RoboDK station: AE1222-2021-GROUP-E09H-RobotMotionPlan.rdk

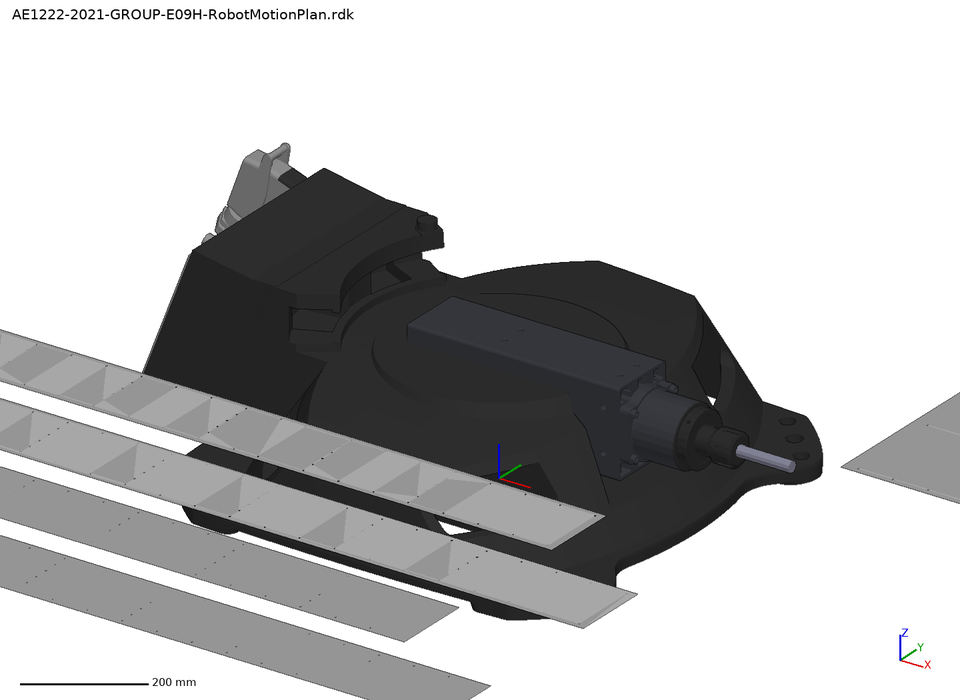
[picture v0: the station drawn from its stored meshes, robots at their saved joint values, targets as dots, program paths as lines]
Station Final (saved by RoboDK 5.2.3). Poses are relative to the parent item; angles as X-Y-Z fixed-axis rotations.
  - frame KUKA KR 210 R2700 extra Base at (0, 0, 0) mm
    - robot KUKA KR 210 R2700 extra: 6 axes, payload 210 kg, reach 2696 mm, repeatability 0.06 mm, weight 1068 kg
        joint limits [-185, -140, -120, -350, -125, -350] to [185, -5, 155, 350, 125, 350]; home [0, -90, 90, 0, 0, 0]; saved at [81.28, -116.082, 145.473, 263.789, 78.817, -240.018]
      - tool Spindle, TCP at (557.2, 0, 176) mm, rotated rx 0 ry 90 rz 0 deg, size 692.9 x 170 x 256 mm
  - Python program Plan, spread panels (listed below)
  - object Panel_Root_Bottom at (1000, 901.6, 500) mm, rotated rx 180 ry 0 rz 0 deg, size 1500 x 400 x 0.8 mm, geometry from Panel_Root_Bottom.stl
  - object Panel_Root_Top at (1000, 1400, 500) mm, rotated rx 180 ry 0 rz 0 deg, size 1500 x 400 x 0.8 mm, geometry from Panel_Root_Top.stl
  - object Panel_Tip - Bottom at (1000, 0, 500) mm, rotated rx 180 ry 0 rz -180 deg, size 1500 x 400 x 0.8 mm, geometry from Panel_Tip - Bottom.stl
  - object Panel_Tip - Top at (1000, -500, 500) mm, rotated rx 180 ry 0 rz -180 deg, size 1500 x 400 x 0.8 mm, geometry from Panel_Tip - Top.stl
  - object Side_Panel_Root_Long at (-500, -1600, 500) mm, rotated rx 0 ry -90 rz -90 deg, size 0.8 x 1500 x 148.4 mm, geometry from Side_Panel_Root_Long.stl
  - object Side_Panel_Root_Short at (-500, -1400, 500) mm, rotated rx 0 ry -90 rz -90 deg, size 0.8 x 1300 x 148.4 mm, geometry from Side_Panel_Root_Short.stl
  - object Side_Panel_Tip_Long at (-500, -1200, 500) mm, rotated rx 0 ry 90 rz 90 deg, size 0.8 x 1500 x 148.4 mm, geometry from Side_Panel_Tip_Long.stl
  - object Side_Panel_Tip_Short at (-500, -1000, 500) mm, rotated rx 0 ry 90 rz 90 deg, size 0.8 x 1300 x 148.4 mm, geometry from Side_Panel_Tip_Short.stl

--- Python program Plan, spread panels ---
from robolink import *
from robodk import *
import time




data = open('AE1222-2021-GROUP-E09H-CoordinateFile-PanelRootBottom.txt')






# read table and get rid of fat
x = 1000
y = 1000
z = 500


table = []
test = []

for line in data:
    row = line.split('\t')
    for i in range(7):
        del row[-1]
    res = [float(i) for i in row]
    res[0] += x
    res[1] += y
    res[2] += z
    table.append(res)
print(table)




RDK = Robolink()


RDK.Render(False)


list_items = RDK.ItemList()
for item in list_items:
    if item.Name().startswith('Auto'):
        item.Delete()


robot = RDK.ItemUserPick('Select a robot', ITEM_TYPE_ROBOT)
robot.setSpeed(500)

RDK.Render(True)


if not robot.Valid():
    quit()


reference = robot.Parent()


robot.setPoseFrame(reference)


pose_ref = robot.Pose()
print(Pose_2_TxyzRxyz(pose_ref))

pose_i = pose_ref
pose_i.setPos(table[0])
robot.MoveJ(pose_i)

for i in range(len(table)-1):

    pose_i = pose_ref
    pose_i.setPos(table[i+1])


    robot.MoveL(pose_i)


data = open('AE1222-2021-GROUP-E09H-CoordinateFile-PanelRootTop.txt')






# read table and get rid of fat
x = 1000
y = 500
z = 500


table = []
test = []

for line in data:
    row = line.split('\t')
    for i in range(7):
        del row[-1]
    res = [float(i) for i in row]
    res[0] += x
    res[1] += y
    res[2] += z
    table.append(res)
print(table)




RDK = Robolink()


RDK.Render(False)


list_items = RDK.ItemList()
for item in list_items:
    if item.Name().startswith('Auto'):
        item.Delete()


robot = RDK.ItemUserPick('Select a robot', ITEM_TYPE_ROBOT)


RDK.Render(True)


if not robot.Valid():
    quit()


reference = robot.Parent()


robot.setPoseFrame(reference)


pose_ref = robot.Pose()
print(Pose_2_TxyzRxyz(pose_ref))





for i in range(len(table)):

    pose_i = pose_ref
    pose_i.setPos(table[i])


    robot.MoveL(pose_i)




data = open('AE1222-2021-GROUP-E09H-CoordinateFile-PanelTipBottom.txt')






# read table and get rid of fat
x = 1000
y = 0
z = 500


table = []
test = []

for line in data:
    row = line.split('\t')
    for i in range(7):
        del row[-1]
    res = [float(i) for i in row]
    res[0] += x
    res[1] += y
    res[2] += z
    table.append(res)
print(table)




RDK = Robolink()


RDK.Render(False)


list_items = RDK.ItemList()
for item in list_items:
    if item.Name().startswith('Auto'):
        item.Delete()


robot = RDK.ItemUserPick('Select a robot', ITEM_TYPE_ROBOT)


RDK.Render(True)


if not robot.Valid():
    quit()


reference = robot.Parent()


robot.setPoseFrame(reference)


pose_ref = robot.Pose()
print(Pose_2_TxyzRxyz(pose_ref))


pose_i = pose_ref
pose_i.setPos(table[0])
robot.MoveJ(pose_i)

for i in range(len(table)-1):

    pose_i = pose_ref
    pose_i.setPos(table[i+1])


    robot.MoveL(pose_i)




data = open('AE1222-2021-GROUP-E09H-CoordinateFile-PanelTipTop.txt')






# read table and get rid of fat
x = 1000
y = -500
z = 500


table = []
test = []

for line in data:
    row = line.split('\t')
    for i in range(7):
        del row[-1]
    res = [float(i) for i in row]
    res[0] += x
    res[1] += y
    res[2] += z
    table.append(res)
print(table)




RDK = Robolink()


RDK.Render(False)


list_items = RDK.ItemList()
for item in list_items:
    if item.Name().startswith('Auto'):
        item.Delete()


robot = RDK.ItemUserPick('Select a robot', ITEM_TYPE_ROBOT)


RDK.Render(True)


if not robot.Valid():
    quit()


reference = robot.Parent()


robot.setPoseFrame(reference)


pose_ref = robot.Pose()
print(Pose_2_TxyzRxyz(pose_ref))





for i in range(len(table)):

    pose_i = pose_ref
    pose_i.setPos(table[i])


    robot.MoveL(pose_i)


time.sleep(1) # _______________________________________________________________

data = open('AE1222-2021-GROUP-E09H-CoordinateFile-SidePanelRootLong.txt')






# read table and get rid of fat
x = -500
y = -1600
z = 500


table = []
test = []

for line in data:
    row = line.split('\t')
    for i in range(8):
        del row[-1]
    res = [float(i) for i in row]
    res[0] += x
    res[1] += y
    res[2] += z
    table.append(res)
print(table)




RDK = Robolink()


RDK.Render(False)


list_items = RDK.ItemList()
for item in list_items:
    if item.Name().startswith('Auto'):
        item.Delete()


robot = RDK.ItemUserPick('Select a robot', ITEM_TYPE_ROBOT)


RDK.Render(True)


if not robot.Valid():
    quit()


reference = robot.Parent()


robot.setPoseFrame(reference)


pose_ref = robot.Pose()
print(Pose_2_TxyzRxyz(pose_ref))





for i in range(len(table)):

    pose_i = pose_ref
    pose_i.setPos(table[i])


    robot.MoveL(pose_i)




data = open('AE1222-2021-GROUP-E09H-CoordinateFile-SidePanelRootShort.txt')






# read table and get rid of fat
x = -500
y = -1400
z = 500


table = []
test = []

for line in data:
    row = line.split('\t')
    for i in range(8):
        del row[-1]
    res = [float(i) for i in row]
    res[0] += x
    res[1] += y
    res[2] += z
    table.append(res)
print(table)




RDK = Robolink()


RDK.Render(False)


list_items = RDK.ItemList()
for item in list_items:
    if item.Name().startswith('Auto'):
        item.Delete()


robot = RDK.ItemUserPick('Select a robot', ITEM_TYPE_ROBOT)


RDK.Render(True)


if not robot.Valid():
    quit()


reference = robot.Parent()


robot.setPoseFrame(reference)


pose_ref = robot.Pose()
print(Pose_2_TxyzRxyz(pose_ref))





for i in range(len(table)):

    pose_i = pose_ref
    pose_i.setPos(table[i])


    robot.MoveL(pose_i)




data = open('AE1222-2021-GROUP-E09H-CoordinateFile-SidePanelTipLong.txt')






# read table and get rid of fat
x = -500
y = -1200
z = 500


table = []
test = []

for line in data:
    row = line.split('\t')
    for i in range(8):
        del row[-1]
    res = [float(i) for i in row]
    res[0] += x
    res[1] += y
    res[2] += z
    table.append(res)
print(table)




RDK = Robolink()


RDK.Render(False)


list_items = RDK.ItemList()
for item in list_items:
    if item.Name().startswith('Auto'):
        item.Delete()


robot = RDK.ItemUserPick('Select a robot', ITEM_TYPE_ROBOT)


RDK.Render(True)


if not robot.Valid():
    quit()


reference = robot.Parent()


robot.setPoseFrame(reference)


pose_ref = robot.Pose()
print(Pose_2_TxyzRxyz(pose_ref))





for i in range(len(table)):

    pose_i = pose_ref
    pose_i.setPos(table[i])


    robot.MoveL(pose_i)




data = open('AE1222-2021-GROUP-E09H-CoordinateFile-SidePanelTipShort.txt')






# read table and get rid of fat
x = -500
y = -1000
z = 500


table = []
test = []

for line in data:
    row = line.split('\t')
    for i in range(8):
        del row[-1]
    res = [float(i) for i in row]
    res[0] += x
    res[1] += y
    res[2] += z
    table.append(res)
print(table)




RDK = Robolink()


RDK.Render(False)


list_items = RDK.ItemList()
for item in list_items:
    if item.Name().startswith('Auto'):
        item.Delete()


robot = RDK.ItemUserPick('Select a robot', ITEM_TYPE_ROBOT)


RDK.Render(True)


if not robot.Valid():
    quit()


reference = robot.Parent()


robot.setPoseFrame(reference)


pose_ref = robot.Pose()
print(Pose_2_TxyzRxyz(pose_ref))





for i in range(len(table)):

    pose_i = pose_ref
    pose_i.setPos(table[i])


    robot.MoveL(pose_i)


quit()
